INTERFACE IFlush

METHOD Flush : BOOL
VAR_INPUT
END_VAR
END_METHOD

PROPERTY pEndFeedback : BOOL
GET
END_GET
END_PROPERTY

END_INTERFACE

(* stored: Version 1.1.0.1, ProductVersion 3.1.4024.0
   Itf IFlush: Id {46f4c250-ff2e-47f6-91cc-1a4eca9b162c}
   Method Flush: Id {c36b7eed-361a-483d-bc3e-89303fb63d7e}
   Property pEndFeedback: Id {61bb2440-1087-4dbb-aa9e-f872a47e78c6}
   Get Get: Id {396036eb-2ae3-4c28-8d86-8d5854b5bb35} *)
